Staubli VAL3: merge1dNum.pgx

public program merge1dNum(num& x_nNum1[], num& x_nNum2[], num& x_nMerged[])
  local num l_nIndex
  local num i
begin

  resize(x_nMerged,1,size(x_nNum1)+size(x_nNum2))
  call empty1dNum(x_nMerged)

  for l_nIndex=0 to size(x_nNum1)-1
    x_nMerged[i]=x_nNum1[l_nIndex]
    i=i+1
  endFor

  for l_nIndex=0 to size(x_nNum2)-1
    x_nMerged[i]=x_nNum2[l_nIndex]
    i=i+1
  endFor

end
